TYPE DUT_Sensor :
STRUCT
    fCntsInEGU:			REAL;
    {attribute 'pytmc' := '
        pv: EU
        io: i
    '}
    sEGU:				STRING;
    sName:				STRING;
    {attribute 'pytmc' := '
        pv: VALUE
        io: i
    '}
    fValue:				REAL;
    {attribute 'pytmc' := '
        pv: RAWCOUNTS
        io: i
    '}
    iRawCnts AT %I*:	INT;
    iOffset:			INT;
END_STRUCT
END_TYPE

(* stored: Version 1.1.0.1, ProductVersion 3.1.4022.18
   DUT DUT_Sensor: Id {5e4e9a12-8121-4b27-a1b4-c219761879b3} *)
